// TwinCAT 3 PLC project PLC1
// ProgramVersion: 3.1.4024.12
// libraries:
//   Tc2_Standard, * (Beckhoff Automation GmbH)
//   Tc2_System, * (Beckhoff Automation GmbH)
//   Tc3_Module, * (Beckhoff Automation GmbH)
// project tree:
//   FBs/Base/ FB_DriveBase.TcPOU
//   FBs/Extended/ FB_DriveCAN.TcPOU, FB_DriveNc.TcPOU (not stored)
//   ITFs/ I_DriveBase.TcIO (not stored)
//   / PlcTask.TcTTO (not stored)
//   POUs/ MAIN.TcPOU (not stored)
// real-time tasks:
//   TASK PlcTask: cycle T#10ms, priority 20, ADS port 350

// ---- FBs/Base/FB_DriveBase.TcPOU
FUNCTION_BLOCK ABSTRACT FB_DriveBase IMPLEMENTS I_DriveBase
VAR
	lrMax : LREAL;
	lrMin : LREAL;
END_VAR

METHOD ABSTRACT Disable : BOOL
END_METHOD

METHOD ABSTRACT Enable : BOOL
END_METHOD

METHOD ABSTRACT MoveToPosition : BOOL
END_METHOD

METHOD ABSTRACT Reset : BOOL
END_METHOD

METHOD SetLimits : BOOL
VAR_INPUT
	lrMax : LREAL;
	lrMin : LREAL;
END_VAR
THIS^.lrMax := lrMax;
THIS^.lrMin := lrMin;
END_METHOD

END_FUNCTION_BLOCK

// ---- FBs/Extended/FB_DriveCAN.TcPOU
FUNCTION_BLOCK FB_DriveCAN EXTENDS FB_DriveBase
VAR_INPUT
END_VAR
VAR_OUTPUT
END_VAR
VAR
END_VAR

METHOD Disable : BOOL
END_METHOD

METHOD Enable : BOOL
END_METHOD

METHOD MoveToPosition : BOOL
END_METHOD

METHOD Reset : BOOL
END_METHOD

END_FUNCTION_BLOCK
